// Mitsubishi GX Works2 project: 0326_timer   PLC: Q03UDV

PROGRAM MAIN
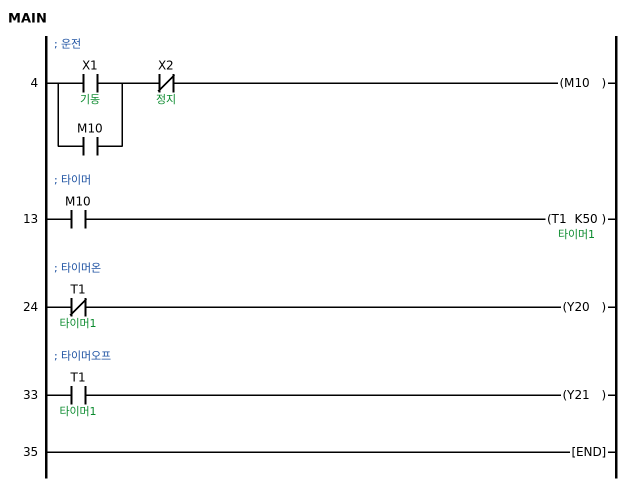
; 운전
4     LD      X1  ; 기동
      OR      M10
      ANI     X2  ; 정지
      OUT     M10
; 타이머
13    LD      M10
      OUT     T1 K50  ; 타이머1
; 타이머온
24    LDI     T1  ; 타이머1
      OUT     Y20
; 타이머오프
33    LD      T1  ; 타이머1
      OUT     Y21
35    END
END_PROGRAM
